TYPE ST_GantryXYZ_Command :
    STRUCT
		ProgramIdRequested : E_RecipeID;
    END_STRUCT
END_TYPE

(* stored: Version 1.1.0.1, ProductVersion 3.1.4024.15
   DUT ST_GantryXYZ_Command: Id {c40493e7-97c3-4ac7-8908-87425e964d7d} *)
